{attribute addProperty BoxType "EL3204-0000-0017"}
{attribute addProperty Id "RTD_Inputs_ChannelAT %I*ARRAY[0..3] OF RTD_Inputs_Channel_B51B79FC32440.50WcStateAT %I*WcState_F855686C1620InfoDataAT %I*InfoData_BC63D37F80100"}
{attribute addProperty CRC "1545010345"}
{attribute addProperty SizeInBites "420"}
{attribute addProperty SizeInBytes "52.5"}
TYPE EL3204_6E5DE158 :
STRUCT
	{attribute addProperty Name "RTD_Inputs_Channel"}
	RTD_Inputs_Channel : ARRAY[0..3] OF RTD_Inputs_Channel_B51B79FC;
	{attribute addProperty Name "WcState"}
	WcState : WcState_F855686C;
	{attribute addProperty Name "InfoData"}
	InfoData : InfoData_BC63D37F;
END_STRUCT
END_TYPE

(* stored: Version 1.2.0.0, ProductVersion 3.1.4024.9
   DUT EL3204_6E5DE158: Id {bef982c8-4fc7-435d-8fc5-f5f91aa22dbb} *)
